// This function has been automatically generated from the project information.
{attribute 'signature_flag' := '1073741824'}
{attribute 'TcGenerated'}
{attribute 'no-analysis'}
FUNCTION F_GetTitle : WSTRING
VAR_INPUT
	
END_VAR

F_GetTitle := "SignalGen";

END_FUNCTION

(* stored: Version 1.1.0.1
   POU F_GetTitle: Id {3e9b6a62-56b1-452c-b566-d2fe29dfdbb8}, SpecialFunc None *)
